% RSLogix 500 project Project5-FINAL.RSS, saved by version 8.30.00.16 %
PROJECT "UNTITLED"    % processor: Bul.1763 MicroLogix 1100 Series B %

PROGRAM FILES
  LAD 2 "MAIN"  3 rungs
  LAD 3 "IO"  5 rungs
  LAD 4 "LOGIC"  1 rungs

DATA FILES
  O0 OUTPUT  4 elements
  I1 INPUT  6 elements
  S2 STATUS  66 elements
  B3 BINARY  3 elements
  T4 TIMER  2 elements
  C5 COUNTER  1 elements
  R6 CONTROL  1 elements
  N7 INTEGER  1 elements
  F8 FLOAT  2 elements

LADDER 2 "MAIN"
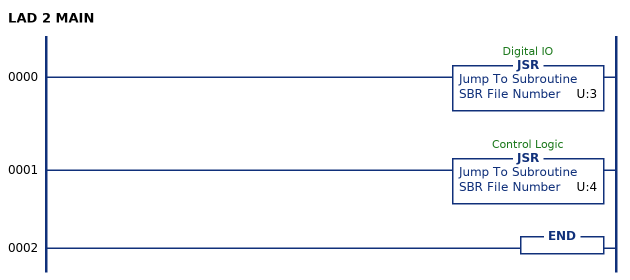
% Rung: 0 %
SOR JSR U:3 EOR
%   U:3  "Digital IO" %
% Rung: 1 %
SOR JSR U:4 EOR
%   U:4  "Control Logic" %
% Rung: 2 %
SOR END EOR

LADDER 3 "IO"
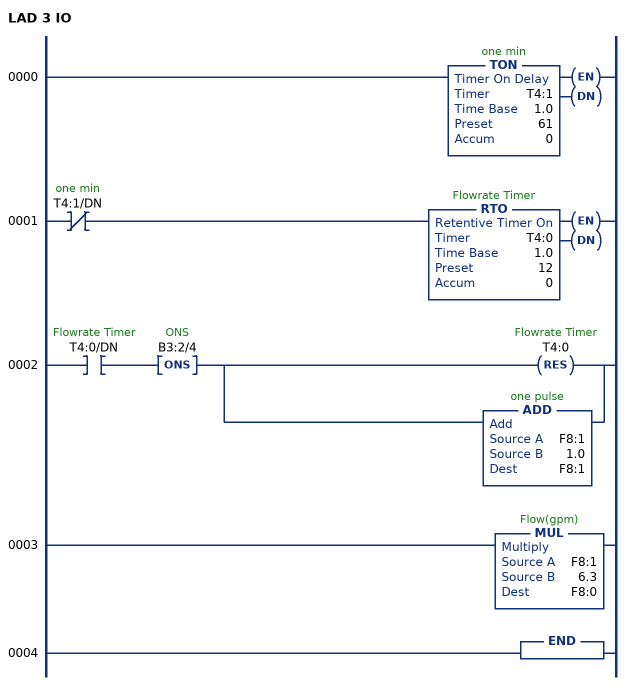
% Rung: 0 %
SOR TON T4:1 1.0 61 0 EOR
%   T4:1  "one min" %
% Rung: 1 %
SOR XIO T4:1/DN RTO T4:0 1.0 12 0 EOR
%   T4:1  "one min" %
%   T4:0  "Flowrate Timer" %
% Rung: 2 %
SOR XIC T4:0/DN ONS B3:2/4 BST RES T4:0 NXB ADD F8:1 1.0 F8:1 BND EOR
%   T4:0  "Flowrate Timer" %
%   B3:2/4  "ONS" %
%   F8:1  "one pulse" %
% Rung: 3 %
SOR MUL F8:1 6.3 F8:0 EOR
%   F8:1  "one pulse" %
%   F8:0  "Flow(gpm)" %
% Rung: 4 %
SOR END EOR

OTHER DOCUMENTED ADDRESSES
  B3:0/1  "START"
  B3:0/2  "START"
  B3:0/3  "START TRIG"
  B3:0/5  "flow DN trigg"
  B3:2/0  "ONS"
  B3:2/1  "ONS"
  B3:2/2  "ONS"
  B3:2/3  "ONS"
  F8:0/1  "pulse"

DATA TABLE (non-zero values as saved)
DATA T4
% .PRE .ACC %
% T4:0 % 12 0
% T4:1 % 61 0
